Fanuc KAREL source: ka00067.KL

-- PROVISIONAL review KL for V940-1; original PC SHA256 8b5bdd6e42ab0ffc991aafaadb39143a5149c6fcb7abdc935fc01dfed44c943e
-- Incomplete behavior may be omitted. Consult companion uncertainty JSON. Do not deploy.
PROGRAM KA00067
%NOLOCKGROUP
-- UNRESOLVED_DECL SRC type=000102
-- UNRESOLVED_DECL DST type=000106
BEGIN
  -- V9_ZERO_TABLE_METADATA_HINT layout=0001; no indexed target words; source/name/runtime held
  -- UNRESOLVED_PC offsets 5-20; opcodes 2E,22,32,35
  -- UNRESOLVED_PC offsets 25-45; opcodes 49,7E,4A
  -- UNRESOLVED_PC offsets 50-54; opcodes 7F
END KA00067
